PROGRAM DistStationControl
VAR
	(* These timers are used to imitate the moving time in the visualization*)
	T1: TIME := TIME#1S0MS;
	T2: TIME := TIME#2000MS;
	TON1: TON;
	TON2: TON;
	TON3: TON;
	TON4: TON;
	TON5: TON;
	TON6: TON;
	
	
	InReset: BOOL; (*  Variable for knowing whether the system is already in reset*)
	
	(* These are just used to maintain the sequence or flow*)
	next1: BOOL;
	next2: BOOL;
END_VAR
VAR // added by the converter: edge detectors and wires of the graphical bodies
    _w1, _w2 : BOOL;
END_VAR

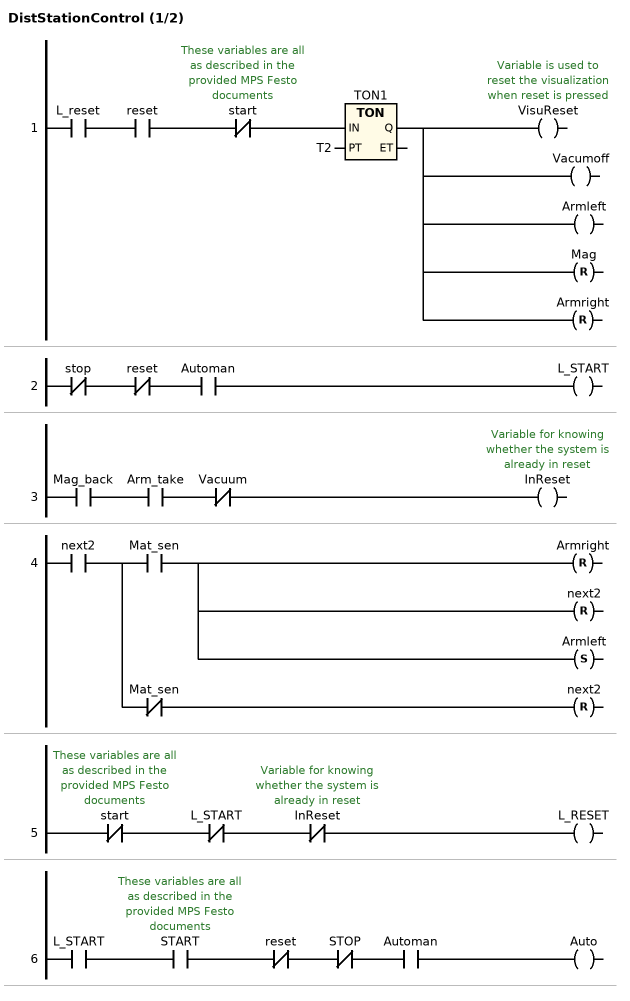
// NETWORK 1
//   start: These variables are all as described in the provided MPS Festo documents
//   VisuReset: Variable is used to reset the visualization when reset is pressed
TON1(IN := L_reset AND reset AND NOT start, PT := T2); // TON
VisuReset := TON1.Q;
Vacumoff := TON1.Q;
Armleft := TON1.Q;
Mag R= TON1.Q;
Armright R= TON1.Q;

// NETWORK 2
L_START := NOT stop AND NOT reset AND Automan;

// NETWORK 3
//   InReset: Variable for knowing whether the system is already in reset
InReset := Mag_back AND Arm_take AND NOT Vacuum;

// NETWORK 4
_w1 := next2;
_w2 := _w1 AND Mat_sen;
Armright R= _w2;
next2 R= _w2;
Armleft S= _w2;
next2 R= _w1 AND NOT Mat_sen;

// NETWORK 5
//   start: These variables are all as described in the provided MPS Festo documents
//   InReset: Variable for knowing whether the system is already in reset
L_RESET := NOT start AND NOT L_START AND NOT InReset;

// NETWORK 6
//   START: These variables are all as described in the provided MPS Festo documents
Auto := (L_START AND START AND NOT reset AND NOT STOP) AND Automan;

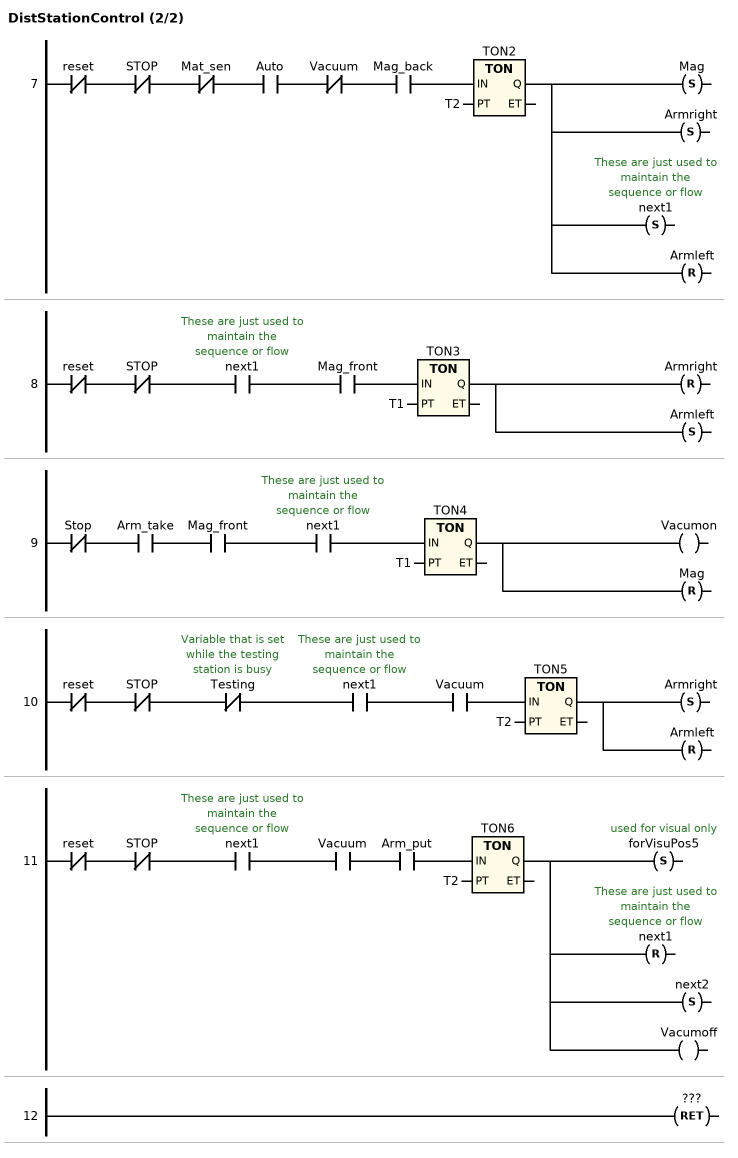
// NETWORK 7
//   next1: These are just used to maintain the sequence or flow
TON2(IN := NOT reset AND NOT STOP AND NOT Mat_sen AND Auto AND NOT Vacuum AND Mag_back, PT := T2); // TON
Mag S= TON2.Q;
Armright S= TON2.Q;
next1 S= TON2.Q;
Armleft R= TON2.Q;

// NETWORK 8
//   next1: These are just used to maintain the sequence or flow
//   T1: These timers are used to imitate the moving time in the visualization
TON3(IN := NOT reset AND NOT STOP AND next1 AND Mag_front, PT := T1); // TON
Armright R= TON3.Q;
Armleft S= TON3.Q;

// NETWORK 9
//   next1: These are just used to maintain the sequence or flow
//   T1: These timers are used to imitate the moving time in the visualization
TON4(IN := NOT Stop AND Arm_take AND Mag_front AND next1, PT := T1); // TON
Vacumon := TON4.Q;
Mag R= TON4.Q;

// NETWORK 10
//   Testing: Variable that is set while the testing station is busy
//   next1: These are just used to maintain the sequence or flow
TON5(IN := NOT reset AND NOT STOP AND NOT Testing AND next1 AND Vacuum, PT := T2); // TON
Armright S= TON5.Q;
Armleft R= TON5.Q;

// NETWORK 11
//   next1: These are just used to maintain the sequence or flow
//   forVisuPos5: used for visual only
TON6(IN := NOT reset AND NOT STOP AND next1 AND Vacuum AND Arm_put, PT := T2); // TON
forVisuPos5 S= TON6.Q;
next1 R= TON6.Q;
next2 S= TON6.Q;
Vacumoff := TON6.Q;

// NETWORK 12
RETURN;

END_PROGRAM

(* stored: Version 1.1.0.1, ProductVersion 3.1.4018.5
   POU DistStationControl: Id {8a5532df-0ba1-4b07-91a7-d9418c6f8dbf}, SpecialFunc None *)
